FUNCTION_BLOCK FB_JointSetup EXTENDS FB_StateMachine IMPLEMENTS  I_StateMachine
VAR_INPUT
	bStart : BOOL;	
	
	stAxis : REFERENCE TO ST_JointAxis;
END_VAR
VAR_OUTPUT
END_VAR
VAR
	eInnerState : E_JointSetupStates;
	bCompleted : BOOL;
	dtTimeCompleted: DATE_AND_TIME;
	bForceSetup : REFERENCE TO BOOL;
	stAbsEncoderAxisRef : REFERENCE TO AXIS_REF;
	stIncEncoderAxisRef : REFERENCE TO AXIS_REF;
	fbAbsEncoderHome : MC_Home;
	fbIncEncoderHome : MC_Home;
END_VAR

OuterLopSM();

METHOD Disable : BOOL
VAR
	bChildBusy  : BOOL := FALSE;
END_VAR
fbAbsEncoderHome(Axis:=stAbsEncoderAxisRef,Execute:=TRUE,HomingMode:=MC_HomingMode.MC_ResetCalibration);
fbIncEncoderHome(Axis:=stIncEncoderAxisRef,Execute:=TRUE,HomingMode:=MC_HomingMode.MC_ResetCalibration);

IF fbAbsEncoderHome.Busy THEN
	bChildBusy := TRUE;
ELSIF fbAbsEncoderHome.Error THEN	
	{warning 'Is below call acceptable here?'}
	fbEventHandler(nBeckhoffID:=fbAbsEncoderHome.ErrorID);
	fbAbsEncoderHome(Axis:=stAbsEncoderAxisRef,Execute:=FALSE);
	bChildBusy := TRUE;
END_IF

IF fbIncEncoderHome.Busy THEN
	bChildBusy := TRUE;
ELSIF fbIncEncoderHome.Error THEN	
	{warning 'Is below call acceptable here?'}
	fbEventHandler(nBeckhoffID:=fbIncEncoderHome.ErrorID);
	fbIncEncoderHome(Axis:=stIncEncoderAxisRef,Execute:=FALSE);
	bChildBusy := TRUE;
END_IF

IF bChildBusy THEN
	Disable := FALSE;
ELSE
	Disable := TRUE;
END_IF
END_METHOD

METHOD InnerLoopSM : BOOL
// update all children FBs
fbAbsEncoderHome(Axis:=stAbsEncoderAxisRef);
fbIncEncoderHome(Axis:=stIncEncoderAxisRef);

CASE CyclicInnerCase(TO_STRING(eInnerState)) OF
	E_JointSetupStates.Idle:
		IF bStart THEN
			bStart := FALSE;
			IF SetupNeeded THEN
				ChangeInnerState(E_JointSetupStates.SetAbsEncoderPositiveDir);
			ELSE
				// Stay in Idle as setup is not needed
			END_IF
		END_IF
		
	E_JointSetupStates.SetAbsEncoderPositiveDir:


		
END_CASE
END_METHOD

METHOD Reset : BOOL
// reset variables specific to this FB 
bCompleted := FALSE;
dtTimeCompleted := DATE_AND_TIME#1970-1-1-0:0:0;

// Reactivate children FBs
//none
END_METHOD

METHOD Setup : BOOL
eStateMachineSourceID := eStateSourceID;
stAbsEncoderAxisRef REF= stAxis.stAbsEncoderAxisRef;
stIncEncoderAxisRef REF= stAxis.stIncEncoderAxisRef;
bForceSetup REF= stAxis.bForceSetup;
SetInnerEnumeration(nStateEnum:=THIS^.eInnerState);
END_METHOD

PROPERTY SetupNeeded : BOOL
GET
// TODO: Check if dtTimeCompleted is too old. If so set SetupNeeded := TRUE
IF bForceSetup THEN
	SetupNeeded := TRUE;
ELSE
	SetupNeeded := NOT bCompleted;
END_IF
END_GET
END_PROPERTY

PROPERTY TimeCompleted : DATE_AND_TIME
GET
TimeCompleted := dtTimeCompleted;
END_GET
END_PROPERTY

END_FUNCTION_BLOCK

(* stored: Version 1.1.0.1, ProductVersion 3.1.4024.12
   POU FB_JointSetup: Id {888c861b-deb3-49aa-a879-accf1d9a1954}, SpecialFunc None
   Folder Properties: Id {5b71f894-4830-45e3-a348-c9d8dfdeb40b}
   Method Disable: Id {97bb9696-0f2a-46f9-97ab-37b590fc03fc}
   Method InnerLoopSM: Id {970bdd2b-e89f-46f7-a0af-71a227ac147c}
   Method Reset: Id {871f704e-650a-46ea-9b4c-7ea6dbb0dbd7}
   Method Setup: Id {70b8979c-e330-4991-a613-d0ceba69cc54}
   Property SetupNeeded: Id {ffb6cc3d-f202-435a-ba65-d363fe30b912}
   Get Get: Id {d7417a21-ce13-46cc-9525-3becc3b92b13}
   Property TimeCompleted: Id {5965413c-fef8-41b3-ae72-1bc57903c58a}
   Get Get: Id {0aa84971-4991-4efe-95bd-4ffd6195aa01} *)
